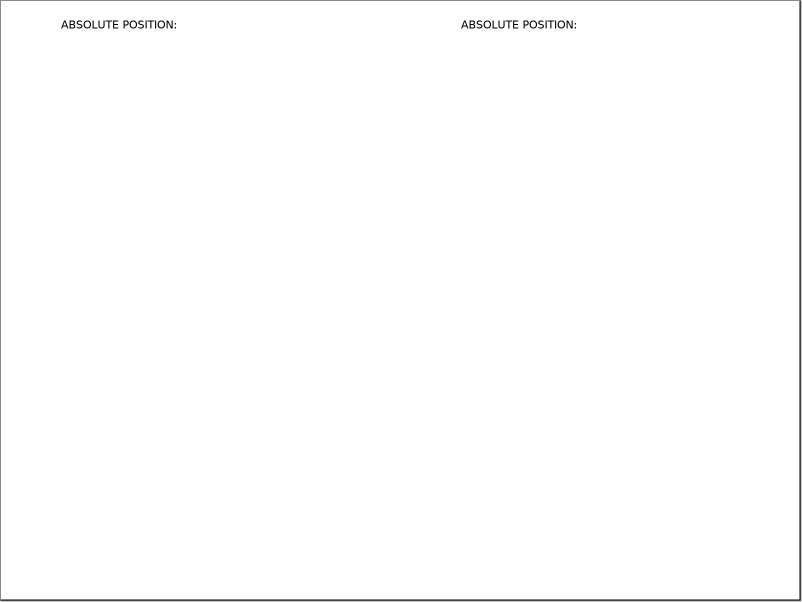
VISUALIZATION F36_Torque_Control  // 802x602
    Rectangle (0,0 800x600)
    Label (10,10 170x30), "ABSOLUTE POSITION:"
    Label (410,10 170x30), "ABSOLUTE POSITION:"
END_VISUALIZATION

(* stored: Version 1.1.0.1, ProductVersion 3.1.4022.7
   Visu F36_Torque_Control: Id {15520fa8-f021-44f8-9548-3091fe5d0249} *)
